// TIA Portal V18 export
// export: Created 2026-06-09T02:47:53.0358177Z, ExportSetting WithDefaults, DisplayName Totally Integrated Automation Portal, DisplayVersion V18, DisplayName TIA Portal Openness, DisplayVersion V18, DisplayName TIA Portal Version Control Interface, DisplayVersion V18, DisplayName STEP 7 Professional, DisplayVersion V18, DisplayName STEP 7 Safety, DisplayVersion V18, DisplayName WinCC Professional, DisplayVersion V18
FUNCTION_BLOCK "Etykieciarka"   // FB3, LAD
{ S7_Optimized_Access := 'TRUE' }
VERSION : 0.1
// stored: AutoNumber true, IsIECCheckEnabled false, IsRetainMemResEnabled false, MemoryReserve 100, SetENOAutomatically false, UDAEnableTagReadback false
BEGIN

REGION Network 1
   // Start przenośnika taśmowego i zapalenie się lampy sygnalizacyjnej.
   // Wyłącznik etykieciarki znajduje się fizycznie na linii produkcyjnej. Stop natomiast w panelu HMI.
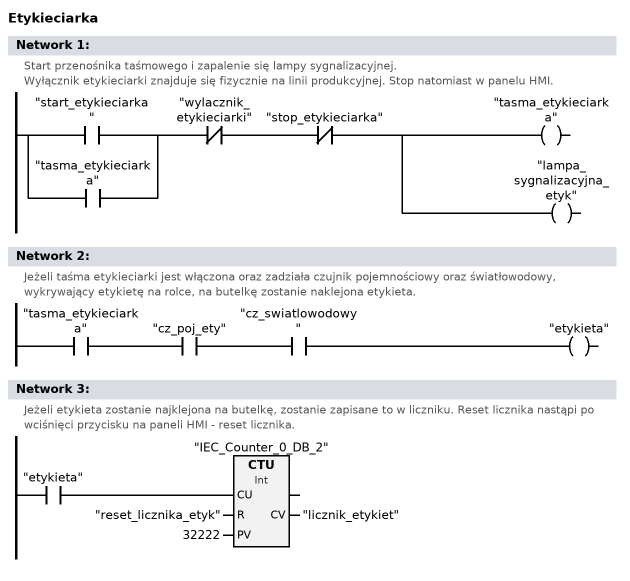
   RUNG wire#powerrail
      Contact( "start_etykieciarka" )
      wire#w1
      I_Contact( "wylacznik_etykieciarki" )
      I_Contact( "stop_etykieciarka" )
      wire#w2
      Coil( "tasma_etykieciarka" )
   END_RUNG
   RUNG wire#powerrail
      Contact( "tasma_etykieciarka" )
   END_RUNG wire#w1
   RUNG wire#w2
      Coil( "lampa_sygnalizacyjna_etyk" )
   END_RUNG
   // the same network as SCL:
   "tasma_etykieciarka" := ("start_etykieciarka" OR "tasma_etykieciarka") AND NOT "wylacznik_etykieciarki" AND NOT "stop_etykieciarka";
   "lampa_sygnalizacyjna_etyk" := "tasma_etykieciarka";
END_REGION

REGION Network 2
   // Jeżeli taśma etykieciarki jest włączona oraz zadziała czujnik pojemnościowy oraz światłowodowy, wykrywający etykietę na rolce, na butelkę zostanie naklejona etykieta.
   RUNG wire#powerrail
      Contact( "tasma_etykieciarka" )
      Contact( "cz_poj_ety" )
      Contact( "cz_swiatlowodowy" )
      Coil( "etykieta" )
   END_RUNG
   // the same network as SCL:
   "etykieta" := "tasma_etykieciarka" AND "cz_poj_ety" AND "cz_swiatlowodowy";
END_REGION

REGION Network 3
   // Jeżeli etykieta zostanie najklejona na butelkę, zostanie zapisane to w liczniku. Reset licznika nastąpi po wciśnięci przycisku na paneli HMI - reset licznika.
   RUNG wire#powerrail
      Contact( "etykieta" )
      { S7_Templates := "value_type := Int" } "IEC_Counter_0_DB_2".CTU(r := "reset_licznika_etyk", pv := 32222, cv => "licznik_etykiet")
   END_RUNG
   // the same network as SCL:
   "IEC_Counter_0_DB_2".CTU(CU := "etykieta", R := "reset_licznika_etyk", PV := 32222, CV => "licznik_etykiet");
END_REGION
END_FUNCTION_BLOCK
